// Mitsubishi GX Works2 project: Domaci zadatak termin2   PLC: FX3S

// task Task_01 (event TRUE, interval 0, priority 31): POU_01

PROGRAM POU_01
VAR
  START : BOOL;
  STOPS : BOOL;
  ukljucen : BOOL;
  TON_1 : TON;
  vreme_t1 : TIME;
  izlaz : BOOL;
  TOF_1 : TOF;
  vreme_t2 : TIME;
  izlaz2 : BOOL;
  CTU_1 : CTU;
  vrednost : INT;
  TON_2 : TON;
  vreme_t3 : TIME;
  brojac : BOOL;
  reset_brojaca : BOOL;
END_VAR
(* structured ladder/FBD written out as ST: instructions are called as NAME(EN, inputs, outputs); _pN, _eN, _tN stand for wires *)
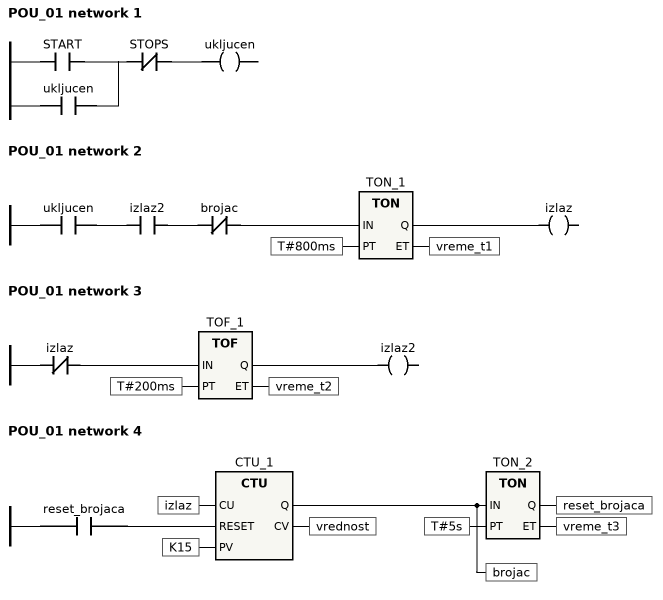
(* network 1 *)
ukljucen := (START OR ukljucen) AND NOT STOPS;
(* network 2 *)
TON_1(IN := ukljucen AND izlaz2 AND NOT brojac, PT := T#800ms, ET => vreme_t1);
izlaz := TON_1.Q;
(* network 3 *)
TOF_1(IN := NOT izlaz, PT := T#200ms, ET => vreme_t2);
izlaz2 := TOF_1.Q;
(* network 4 *)
CTU_1(CU := izlaz, RESET := reset_brojaca, PV := K15, CV => vrednost);
brojac := CTU_1.Q;
TON_2(IN := CTU_1.Q, PT := T#5s, Q => reset_brojaca, ET => vreme_t3);
END_PROGRAM
